// This function has been automatically generated from the project information.
{attribute 'signature_flag' := '1073741824'}
{attribute 'TcGenerated'}
FUNCTION F_GetTitle : WSTRING
VAR_INPUT
	
END_VAR

F_GetTitle := "tclib_ph_lv1_comm_opcua";

END_FUNCTION

(* stored: Version 1.1.0.1, ProductVersion 3.1.4019.2
   POU F_GetTitle: Id {37039e92-e27e-412f-bdf3-f6ca95d19fd9}, SpecialFunc None *)
